{attribute 'qualified_only' := ''}
{attribute 'strict' := ''}
TYPE eAdasKonfig_State :
(
	Init,
	SendTrackConfig,
	WaitForSelectFlag,
	ConfigCurrent
);
END_TYPE

(* stored: Version 1.1.0.1, ProductVersion 3.1.4022.16
   DUT eAdasKonfig_State: Id {799ca86f-9e15-432e-9684-5b36757c892b} *)
